FUNCTION_BLOCK EL3202
VAR
	_io : EL3xx2_Data;
	{attribute addProperty Name "WcState"}
	_wcState : WcStateInputToggle;
	{attribute addProperty Name "Info data"}
	_infoData : InfoDataAds;
END_VAR

PROPERTY IO : REFERENCE TO EL3xx2_Data
GET
IO REF= _io;
END_GET
END_PROPERTY

PROPERTY WcState : REFERENCE TO WcStateInputToggle
GET
WcState REF= _wcState;
END_GET
END_PROPERTY

END_FUNCTION_BLOCK

(* stored: Version 1.1.0.1, ProductVersion 3.1.4024.9
   POU EL3202: Id {f51178d2-0a68-015c-08cf-7d60ed2a4950}, SpecialFunc None
   Property IO: Id {77e67903-3438-08b7-1c7a-e3674ab397f4}
   Get Get: Id {0be61012-6a56-0d77-3e5b-6ee06902e185}
   Property WcState: Id {351ff06f-fbae-0b3c-0bdf-2cff513a2f29}
   Get Get: Id {37961a67-f37e-0d5e-2f85-7be9e4731dc2} *)
